PROGRAM MAIN
VAR
	SampleDevice : UDINT;
END_VAR

SampleDevice := SampleDevice + 1;

END_PROGRAM

(* stored: Version 1.1.0.1, ProductVersion 3.1.4024.4
   POU MAIN: Id {f88a4a61-b782-4030-a966-b2f336fe2bbe}, SpecialFunc None *)
